TYPE E_LibState :
(
	Idle := 0,
	Done := 1
);
END_TYPE

(* stored: Version 1.1.0.1, ProductVersion 3.1.4026.18
   DUT E_LibState: Id {00000000-0000-0000-0000-000000000081} *)
